// TwinCAT 3 PLC project Desktop
// ProgramVersion: 3.1.4024.0
// libraries:
//   Tc2_BABasic, * (Beckhoff Automation GmbH)
//   Tc2_EtherCAT, * (Beckhoff Automation GmbH)
//   Tc2_Math, * (Beckhoff Automation GmbH)
//   Tc2_Standard, * (Beckhoff Automation GmbH)
//   Tc2_System, * (Beckhoff Automation GmbH)
//   Tc2_Utilities, * (Beckhoff Automation GmbH)
//   Tc3_BA2_Common, * (Beckhoff Automation GmbH)
//   Tc3_BA_Common, * (Beckhoff Automation GmbH)
//   Tc3_LS, * (Beckhoff Automation GmbH)
//   Tc3_Module, * (Beckhoff Automation GmbH)
// project tree:
//   General/ SoftwareVersionControl.TcPOU
//   Main/ Eventlogger.TcPOU, E_EventType.TcDUT, FB_CSVPersistentEventStorage.TcPOU, I_PersistentEventStorage.TcIO, ST_Event.TcDUT, UpdateEventTimeStamp.TcPOU, MAIN.TcPOU
//   / PlcTask.TcTTO
//   Testing/ Circle.TcPOU, FB_A.TcPOU, FB_B.TcPOU, F_DeliverType.TcPOU, I_Name.TcIO, Shape.TcIO
// real-time tasks:
//   TASK PlcTask: cycle T#10ms, priority 20, ADS port 350
//   TASK PlcTask1: cycle T#10ms, priority 21, ADS port 351
//   TASK PlcTask2: cycle T#10ms, priority 22, ADS port 352

CONFIGURATION Desktop
    RESOURCE PLC ON TwinCAT3
        TASK PlcTask(INTERVAL := T#10ms, PRIORITY := 20);
        PROGRAM MAIN WITH PlcTask : MAIN;
    END_RESOURCE
END_CONFIGURATION

// ---- Main/E_EventType.TcDUT
{attribute 'qualified_only'}
{attribute 'strict'}
{attribute 'to_string'}
TYPE E_EventType :
(
	Alarm := 0,
	Messages:=1,
	Warning:=2
);
END_TYPE

// ---- Main/ST_Event.TcDUT
TYPE ST_Event :
STRUCT
	eEventTypes: E_EventType;
	eEventSeverity: TcEventSeverity;
	eEventIdentity: UDINT;
	eEventText: STRING(255);
	dtTimestamp: DATE_AND_TIME;	
END_STRUCT
END_TYPE

// ---- Main/I_PersistentEventStorage.TcIO
INTERFACE I_PersistentEventStorage

METHOD StoreEvent
VAR_INPUT
	stEvent:ST_Event;
END_VAR
END_METHOD

END_INTERFACE

// ---- Testing/I_Name.TcIO
INTERFACE I_Name

PROPERTY Name : STRING
GET
END_GET
SET
END_SET
END_PROPERTY

END_INTERFACE

// ---- Testing/Shape.TcIO
INTERFACE Shape

METHOD Area : Float
VAR_INPUT
	fRadiusOfShape: float;
END_VAR
END_METHOD

METHOD Price : float
VAR_INPUT
	fArea : float;
	fPriceOverArea: float;
END_VAR
END_METHOD

PROPERTY PricePerMeter : float
GET
END_GET
SET
END_SET
END_PROPERTY

PROPERTY Radius : float
GET
END_GET
SET
END_SET
END_PROPERTY

END_INTERFACE

// ---- Main/MAIN.TcPOU
PROGRAM MAIN
(***********************************************************************************************************************************************************************************************************************
Company			EclipseAutomation(Penang) Sdn. Bhd					
Project			4 Position Demolding Test System
Author			BC Yeoh
Desciption		Global discription of version library

************************************************************************************************************************************************************************************************************************
Change/DATE			Name				Version			Change desciption
************************************************************************************************************************************************************************************************************************
19 Sep 2023			BC Yeoh				Vx.y.pp			Draft (will update to first release/Qualification version after SAT) 



************************************************************************************************************************************************************************************************************************)
				

VAR
//	Trigger : BOOL;
//	Eventlogger: Eventlogger(CSVPersistentEventStorage);
//	CSVPersistentEventStorage: FB_CSVPersistentEventStorage;
//	eEventTypes1: E_EventType:=E_EventType.Alarm ;
//	eEventSeverity1: TcEventSeverity:= TcEventSeverity.Error;
//	eEventIdentity1: UDINT :=123;
//	eEventText1: STRING(255):= 'What does the fok say';
fCircle : Circle;
fPriceofCircle : float;
    iName     : I_Name;

    fbSampleA : FB_A; 
    sNameA    : STRING;       // will be 'My name is A.'

    fbSampleB : FB_B;
    sNameB    : STRING;       // will be 'My name is B.' after first cycle
                              // and will be 'New name' afterwards
END_VAR

//IF Trigger THEN
//	Eventlogger.AddEvent(eEventTypes1,eEventSeverity1,eEventIdentity1,eEventText1);
//	Trigger:=false;
//END_IF
//CSVPersistentEventStorage();

// Calling axis module by passing input parameter "bExecuteProcess" of this method to the input parameter "bExecute" of method "Execute"
//fCircle.Radius:=
//fCircle.Area(fRadiusOfShape:=10.00);
//fCircle.Price(fArea:=fCircle.
//,fPriceOverArea:=10.00);

//// assign FB instance fbSample1 to interface variable
//iName := fbSampleA;
 
//// access to name property of fbSample1 via interface variable (Get)
//sNameA := iName.Name;
 
//// access to name property of fbSample2 via FB instance (Get and Set)
//sNameB := fbSampleB.Name;
//fbSampleB.Name := 'New name';

END_PROGRAM

// ---- Testing/Circle.TcPOU
FUNCTION_BLOCK Circle IMPLEMENTS Shape
VAR_INPUT
	fPricePM: float;
	fRadius:float;
END_VAR
VAR_OUTPUT
	fFinalPrice:float;
END_VAR
VAR
END_VAR

{warning 'add method implementation '}
METHOD Area : Tc2_Utilities.FLOAT
VAR_INPUT
	fRadiusOfShape	: Tc2_Utilities.FLOAT;
END_VAR
Area:=3.142*fRadiusOfShape*fRadiusOfShape;
END_METHOD

{warning 'add method implementation '}
METHOD Price : Tc2_Utilities.FLOAT
VAR_INPUT
	fArea	: Tc2_Utilities.FLOAT;
	fPriceOverArea	: Tc2_Utilities.FLOAT;
END_VAR
Price:=fArea*fPriceOverArea;
END_METHOD

{warning 'add property implementation'}
PROPERTY PricePerMeter : Tc2_Utilities.FLOAT
GET
END_GET
SET
END_SET
END_PROPERTY

{warning 'add property implementation'}
PROPERTY Radius : Tc2_Utilities.FLOAT
GET
END_GET
SET
END_SET
END_PROPERTY

END_FUNCTION_BLOCK

// ---- Testing/FB_A.TcPOU
FUNCTION_BLOCK FB_A IMPLEMENTS I_Name

VAR
    sVar1 : STRING := 'My name is A.';
END_VAR

{warning 'add property implementation'}
PROPERTY Name : STRING
GET
Name := sVar1;
END_GET
SET
sVar1 := Name;
END_SET
END_PROPERTY

END_FUNCTION_BLOCK

// ---- Testing/FB_B.TcPOU
FUNCTION_BLOCK FB_B IMPLEMENTS I_Name

VAR
    sVar2 : STRING := 'My name is B.'; 
END_VAR

{warning 'add property implementation'}
PROPERTY Name : STRING
GET
Name := sVar2;
END_GET
SET
sVar2 := Name;
END_SET
END_PROPERTY

END_FUNCTION_BLOCK

// ---- General/SoftwareVersionControl.TcPOU
(*****************************************************************************************************

Company			EclipseAutomation(Penang) Sdn. Bhd					
Project			4 Position Demolding Test System
Author			BC Yeoh
Desciption		Global discription of version library
QV-Number		N/A

Used libs		Tc2_Standard	3.3.3.0		 02 Dec 2019 5:54:56 PM			
				Tc2_System		3.5.3.0		 24 Feb 2023 11:18:34 AM
				Tc3_Module		3.3.23.0	 18 Jan 2023 3:34:30 PM
				
				
				
				
				
				
				
Used shortcuts	-CV		CibaVision 				
				-RT		RoundTable/Turning Table
				
				
				
				
				
				
				
****************************************************************************************)
PROGRAM SoftwareVersionControl
VAR
END_VAR

(*****************************************************************************************************
Change/DATE			Name				Version/Change Request Nr			Change desciption
******************************************************************************************************
19 Sep 2023			BC Yeoh				Vx.y.pp/PRxxxxxxxx					Draft (will update to first release/Qualification version after SAT) 
			
				
				
				
				
				
				
****************************************************************************************)

END_PROGRAM

// ---- Main/Eventlogger.TcPOU
FUNCTION_BLOCK Eventlogger
VAR
		Eventbuffer : ARRAY[0..MaxBuffersize] OF ST_Event;
		CurrentBufferIndex : INT :=0;
		_PersistentEventStorage : I_PersistentEventStorage;
END_VAR
VAR CONSTANT
	MaxBuffersize: INT := 100;
END_VAR

METHOD PUBLIC AddEvent : BOOL
VAR_INPUT
	eEventTypes: E_EventType;
	eEventSeverity: TcEventSeverity;
	eEventIdentity: UDINT;
	eEventText: STRING(255);
END_VAR
IF NOT IsEventBufferFull() THEN
	CurrentBufferIndex:=CurrentBufferIndex+1;
	Eventbuffer[CurrentBufferIndex].eEventTypes:=eEventTypes;
	Eventbuffer[CurrentBufferIndex].eEventSeverity:=eEventSeverity;
	Eventbuffer[CurrentBufferIndex].eEventIdentity:=eEventIdentity;
	Eventbuffer[CurrentBufferIndex].eEventText:=eEventText;
	UpdateEventTimeStamp(stEvent:=Eventbuffer[CurrentBufferIndex]);
	AddEvent:= TRUE;
ELSE
	AddEvent:= FALSE;
END_IF

//Store the event here
_PersistentEventStorage.StoreEvent(stEvent := Eventbuffer[CurrentBufferIndex]);
END_METHOD

METHOD FB_init : BOOL
VAR_INPUT
	bInitRetains : BOOL; // if TRUE, the retain variables are initialized (warm start / cold start)
	bInCopyCode : BOOL;  // if TRUE, the instance afterwards gets moved into the copy code (online change)
	iPersistentEventStorage:I_PersistentEventStorage;
END_VAR
_PersistentEventStorage:=iPersistentEventStorage;
END_METHOD

METHOD PRIVATE IsEventBufferFull : BOOL
IF (CurrentBufferIndex+1)> MaxBuffersize THEN
	IsEventBufferFull:=TRUE;
ELSE
	IsEventBufferFull:=FALSE;		
END_IF
END_METHOD

END_FUNCTION_BLOCK

// ---- Main/UpdateEventTimeStamp.TcPOU
FUNCTION UpdateEventTimeStamp : ST_Event
VAR_INPUT
	stEvent : REFERENCE TO ST_Event ;
END_VAR

VAR
	fbgetsystemtime: GETSYSTEMTIME;
	stFileTime : T_FILETIME;
	nHigh : UDINT;
	nLow : UDINT;	
END_VAR

fbgetsystemtime(timeLodw=>stFileTime.dwLowDateTime , timeHidw=>stFileTime.dwHighDateTime); 

stEvent.dtTimestamp:=FILETIME_TO_DT(stFileTime);

END_FUNCTION

// ---- Main/FB_CSVPersistentEventStorage.TcPOU
FUNCTION_BLOCK FB_CSVPersistentEventStorage IMPLEMENTS I_PersistentEventStorage
VAR
	eWriteState : (File_Open_Trigger,File_Open,Wait_For_Event,Write_Event_Trigger,Write_Event,File_Close_Trigger,File_Close,Error);
	fbFileOpen:FB_FileOpen:= (sPathName:= 'C:\Users\Beckhoff\Desktop\Event.log',nMode:=FOPEN_MODEAPPEND OR FOPEN_MODETEXT);
	fbFilePuts: FB_FilePuts;
//	fbFileWrite:FB_FileWrite;
	fbFileClose:FB_FileClose;
	stEventWrittenToFile:ST_Event;
	CSVString:T_MaxString;
END_VAR

CASE eWriteState OF
	File_Open_Trigger:
		fbFileOpen(bExecute:=TRUE);
		eWriteState:=File_Open;
		
	File_Open:
		fbFileOpen(bExecute:=FALSE);
		IF fbFileOpen.bError THEN
			eWriteState:=Error;
		ELSIF NOT fbFileOpen.bBusy AND fbFileOpen.hFile<>0 THEN
			eWriteState:=Wait_For_Event;
		END_IF;
		
	Wait_For_Event:
	//do nothing
	
	Write_Event_Trigger:
		CSVString:=CreateCSVString(stEvent:=stEventWrittenToFile);
		fbFilePuts(bExecute:=TRUE,sLine:=CSVString,hFile:=fbFileOpen.hFile);
		eWriteState:=Write_Event;	

	Write_Event:
		fbFilePuts(bExecute:=FALSE);
		IF fbFilePuts.bError THEN
			eWriteState:=Error;
		ELSIF NOT fbFilePuts.bBusy THEN
			eWriteState:=File_Close_Trigger;
		END_IF;
	File_Close_Trigger:
		fbFileClose(bExecute:=TRUE,hFile:=fbFileOpen.hFile);
		eWriteState:=File_Close;	
	File_Close:
		fbFileClose(bExecute:=FALSE);
		IF fbFileClose.bError THEN
			eWriteState:=Error;
		ELSIF NOT fbFileClose.bBusy THEN
			eWriteState:=File_Open_Trigger;
		END_IF;	
END_CASE;

METHOD PRIVATE CreateCSVString : T_MaxString
VAR_INPUT
	stEvent : REFERENCE TO ST_Event;
END_VAR
VAR
	TempString : T_MaxString;
END_VAR

TempString:= TO_STRING(stEvent.eEventTypes);
TempString:=Concat(STR1:= TempString,STR2:=',');
TempString:=Concat(STR1:= TempString,STR2:=TO_STRING(stEvent.eEventSeverity));
TempString:=Concat(STR1:= TempString,STR2:=',');
TempString:=Concat(STR1:= TempString,STR2:=TO_STRING(stEvent.eEventIdentity));
TempString:=Concat(STR1:= TempString,STR2:=',');
TempString:=Concat(STR1:= TempString,STR2:=stEvent.eEventText);
TempString:=Concat(STR1:= TempString,STR2:=',');
TempString:=Concat(STR1:= TempString,STR2:=TO_STRING(stEvent.dtTimestamp));
TempString:=Concat(STR1:= TempString,STR2:='$N');

CreateCSVString:=TempString;
END_METHOD

{warning 'add method implementation '}
METHOD StoreEvent
VAR_INPUT
	stEvent	: ST_Event;
END_VAR
//write csv code
IF eWriteState=Wait_For_Event THEN
	stEventWrittenToFile:=stEvent;
	eWriteState:= Write_Event_Trigger;
END_IF
END_METHOD

END_FUNCTION_BLOCK

// ---- Testing/F_DeliverType.TcPOU
FUNCTION F_DeliverType : string
VAR_INPUT
	iSample : I_Name;
END_VAR

F_DeliverType := iSample.GetType();

END_FUNCTION
